(* Schneider Machine Expert - Basic project 2pompe_alternanza, file version 3.0.0.0 *)
(* ProjectInformations: Name=New project *)

HARDWARE
  Cpu 0: TM221C40R
  EthernetConfiguration: NetworkName=M221, IpAllocationMode=FixedAddress, IpAddress=0.0.0.0, SubnetMask=0.0.0.0
  SerialLineConfiguration: Baud=Baud19200, Parity=ParityEven, DataBits=DataBits8, StopBits=StopBits1, PhysicalMedium=PhysicalMediumRs485, TransmissionMode=TransmissionModeModbusRtu, SlaveId=1, Addressing=SlaveAddressing
  MastTask: UsePeriodScanMode=false, PeriodScan=100
  FastTask: Period=255
  CpuBehavior: StartingMode=StartAsPreviousState, AutoSaveRamOnEeprom=true, WatchdogPeriod=250

SYMBOLS  (address, symbol, comment, settings)
  %M0       P1_USABILE
  %M1       P2_USABILE
  %MW0      ULTIMA_POMPA_CMD
  %I0.0     P1_AUTO
  %I0.1     P1_MOTO
  %I0.2     P1_ANOMALIA
  %I0.3     P2_AUTO
  %I0.4     P2_MOTO
  %I0.5     P2_ANOMALIA
  %I0.6     LVL_MIN
  %I0.7     LVL_MAX
  %Q0.0     P1_CMD
  %Q0.1     P2_CMD

POU New POU
  (* SectionNumber=1 *)

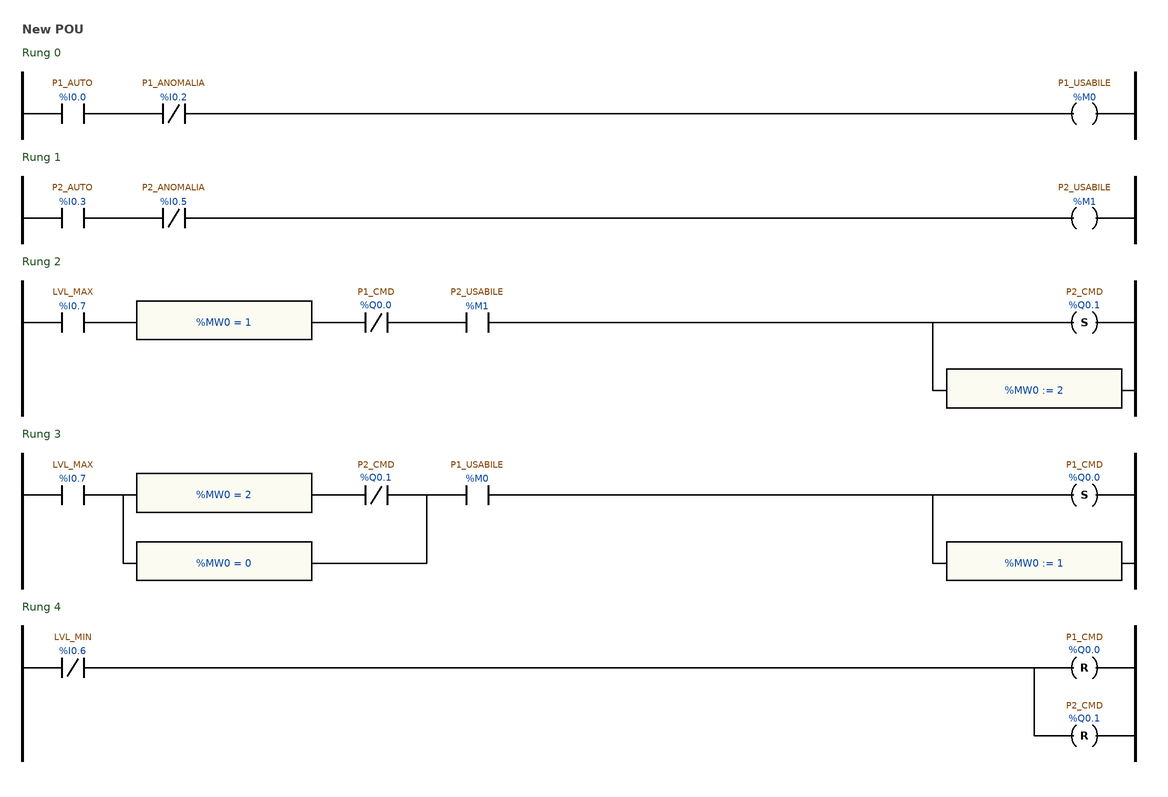

// Rung 0
  LD %I0.0                (* P1_AUTO *)
  ANDN %I0.2              (* P1_ANOMALIA *)
  ST %M0                  (* P1_USABILE *)
  // as ST:
  //   P1_USABILE := P1_AUTO AND NOT P1_ANOMALIA;

// Rung 1
  LD %I0.3                (* P2_AUTO *)
  ANDN %I0.5              (* P2_ANOMALIA *)
  ST %M1                  (* P2_USABILE *)
  // as ST:
  //   P2_USABILE := P2_AUTO AND NOT P2_ANOMALIA;

// Rung 2
  LD %I0.7                (* LVL_MAX *)
  AND [ %MW0 = 1 ]        (* ULTIMA_POMPA_CMD *)
  ANDN %Q0.0              (* P1_CMD *)
  AND %M1                 (* P2_USABILE *)
  S %Q0.1                 (* P2_CMD *)
  [ %MW0 := 2 ]           (* ULTIMA_POMPA_CMD *)
  // as ST:
  //   IF LVL_MAX AND ULTIMA_POMPA_CMD = 1 AND NOT P1_CMD AND P2_USABILE THEN P2_CMD := TRUE; END_IF;
  //   IF LVL_MAX AND ULTIMA_POMPA_CMD = 1 AND NOT P1_CMD AND P2_USABILE THEN ULTIMA_POMPA_CMD := 2; END_IF;

// Rung 3
  LD %I0.7                (* LVL_MAX *)
  AND( [ %MW0 = 2 ]       (* ULTIMA_POMPA_CMD *)
  ANDN %Q0.1              (* P2_CMD *)
  OR [ %MW0 = 0 ]         (* ULTIMA_POMPA_CMD *)
  )
  AND %M0                 (* P1_USABILE *)
  S %Q0.0                 (* P1_CMD *)
  [ %MW0 := 1 ]           (* ULTIMA_POMPA_CMD *)
  // as ST:
  //   IF LVL_MAX AND (ULTIMA_POMPA_CMD = 2 AND NOT P2_CMD OR ULTIMA_POMPA_CMD = 0) AND P1_USABILE THEN P1_CMD := TRUE; END_IF;
  //   IF LVL_MAX AND (ULTIMA_POMPA_CMD = 2 AND NOT P2_CMD OR ULTIMA_POMPA_CMD = 0) AND P1_USABILE THEN ULTIMA_POMPA_CMD := 1; END_IF;

// Rung 4
  LDN %I0.6               (* LVL_MIN *)
  R %Q0.0                 (* P1_CMD *)
  R %Q0.1                 (* P2_CMD *)
  // as ST:
  //   IF NOT LVL_MIN THEN P1_CMD := FALSE; END_IF;
  //   IF NOT LVL_MIN THEN P2_CMD := FALSE; END_IF;
